FUNCTION_BLOCK FB_HumiditySensor EXTENDS FB_Sensor
VAR_INPUT
END_VAR
VAR_OUTPUT
	fHumidity : REAL; //measured relative humidity
END_VAR
VAR
	//I/O-Links
	humidity_IN AT %I* : INT;
	
END_VAR

METHOD GetState_AI : BOOL
VAR_INPUT
END_VAR
//Humidity := (humidity_IN / 32767.0)- Offset 10% ;
fHumidity := (humidity_IN / 32767.0)-0.1;

(*Umrechnungsfaktor muss noch angepasst werden
0 ist minimaler Wert	:= 0 V -> 0 % Luftfeuchtigkeit
32767 ist maximaler Wert := 10 V -> 100 % Luftfeuchtigkeit
*)

//sensor state
sensorState.fValue := fHumidity;
sensorState.sUnit := 'percent';
END_METHOD

END_FUNCTION_BLOCK

(* stored: Version 1.1.0.1, ProductVersion 3.1.4024.6
   POU FB_HumiditySensor: Id {22fdbe35-8890-4e7c-a1dd-a8b878c27712}, SpecialFunc None
   Method GetState_AI: Id {b1aeeb65-9d07-41ad-a773-764ead2b4c78} *)
